TYPE ST_Feeding :
STRUCT
		Info		: ST_FeedingDataInfo;
		Feeback		: ST_FeedingDataFeeback;
		Handshake	: ST_HandshakeBase;
END_STRUCT
END_TYPE

(* stored: Version 1.1.0.1, ProductVersion 3.1.4024.13
   DUT ST_Feeding: Id {d7d18286-bb4a-46cc-861f-1141a410c067} *)
